VAR_GLOBAL
END_VAR

(* stored: Version 1.1.0.1, ProductVersion 3.1.0.23
   GVL MER_CmdState: Id {65c5dc44-bfad-4f14-a5b2-d31766de47b8} *)
